// TwinCAT 3 PLC project IO_Main_Task
// ProgramVersion: 3.1.4026.19
// libraries:
//   Tc2_Standard, * (Beckhoff Automation GmbH)
//   Tc2_System, * (Beckhoff Automation GmbH)
//   Tc3_Module, * (Beckhoff Automation GmbH)
// project tree:
//   DUTs/EtherCAT模組/ EL1409.TcDUT, Murr_IMPACT67.TcDUT, EL2409.TcDUT
//   DUTs/ In_16_To_PLC.TcDUT, Out_16_To_PLC.TcDUT
//   GVLs/ EtherCAT.TcGVL, MainIO.TcGVL
//   / IO_Task.TcTTO
//   POUs/IO轉換/ AI_force.TcPOU, IO_force.TcPOU
//   POUs/IO轉換/控制櫃/ Mod101.TcPOU, Mod401.TcPOU, Mod102.TcPOU, Mod103.TcPOU, Mod104.TcPOU, Mod105.TcPOU, Mod106.TcPOU, Mod107.TcPOU, Mod108.TcPOU, Mod109.TcPOU
//   POUs/ MAIN.TcPOU
// (motion and I/O tree: see PLC project main)
// real-time tasks:
//   TASK Main_IO_Task: cycle T#2ms, priority 6, ADS port 353
//   TASK PlcTask: cycle T#10ms, priority 14, ADS port 350
//   TASK Conveyor: cycle T#10ms, priority 22, ADS port 355
// variable links:

CONFIGURATION IO_Main_Task
    RESOURCE PLC ON TwinCAT3
        TASK IO_Task(INTERVAL := T#2ms, PRIORITY := 6);
        PROGRAM MAIN WITH IO_Task : MAIN;
    END_RESOURCE
END_CONFIGURATION

// ---- DUTs/EtherCAT模組/EL1409.TcDUT
TYPE EL1409 :
STRUCT
	ModType : STRING := 'EL1409';
	Input AT %I*:ARRAY [1..16] OF BOOL;
	WcState AT %I*:BOOL;
	InputToggle AT %I*:BOOL;
	State AT %I*:UINT;
END_STRUCT
END_TYPE

// ---- DUTs/EtherCAT模組/Murr_IMPACT67.TcDUT
TYPE Murr_IMPACT67 :
STRUCT
	ModType : STRING := 'Murr IMPACT67';
	
	Input AT %I*:UINT;
	
	Output AT %Q*:UINT;
	
	Io_State AT %I*:ARRAY[0..7] OF USINT;
	
	WcState AT %I*:BOOL;
	InputToggle AT %I*:BOOL;
	State AT %I*:UINT;
END_STRUCT
END_TYPE

// ---- DUTs/EtherCAT模組/EL2409.TcDUT
TYPE EL2409 :
STRUCT
	ModType : STRING := 'EL2409';
	WcState AT %I*:BOOL;
	State AT %I*:UINT;
	
	Output AT %Q*:ARRAY [1..16] OF BOOL;
END_STRUCT
END_TYPE

// ---- DUTs/In_16_To_PLC.TcDUT
TYPE In_16_To_PLC :
STRUCT
	In AT %Q*:ARRAY [1..16] OF BOOL;
END_STRUCT
END_TYPE

// ---- DUTs/Out_16_To_PLC.TcDUT
TYPE Out_16_To_PLC :
STRUCT
	Out AT %I*:ARRAY [1..16] OF BOOL;
END_STRUCT
END_TYPE

// ---- GVLs/EtherCAT.TcGVL
{attribute 'qualified_only'}
VAR_GLOBAL
	// 主控制櫃 控制器
	MainMod_1 :EL1409;
	MainMod_2 :EL1409;
	MainMod_3 :EL1409;
	MainMod_4 :EL1409;
	MainMod_5 :EL1409;
	MainMod_6 :EL1409;
	MainMod_7 :EL2409;
	MainMod_8 :EL2409;
	MainMod_9 :EL2409;
	
	Murr_Mod : Murr_IMPACT67;
END_VAR

// ---- GVLs/MainIO.TcGVL
{attribute 'qualified_onlY0'}
VAR_GLOBAL
	//
	IO101: In_16_To_PLC;
	//
	IO102: In_16_To_PLC;
	//
	IO103: In_16_To_PLC;
	//
	IO104: In_16_To_PLC;
	//
	IO105: In_16_To_PLC;
	//
	IO106: In_16_To_PLC;
	//
	IO107: Out_16_To_PLC;
	//
	IO108: Out_16_To_PLC;
	//
	IO109: Out_16_To_PLC;
	
	//
	IO401: In_16_To_PLC;
	

	IO101_s : WORD;
	IO102_s : WORD;
	IO103_s : WORD;
	IO104_s : WORD;
	IO105_s : WORD;
	IO106_s : WORD;
	IO107_s : WORD;
	IO108_s : WORD;
	IO109_s : WORD;
	
	IO401_s : WORD;
	
	IO101_f : WORD;
	IO102_f : WORD;
	IO103_f : WORD;
	IO104_f : WORD;
	IO105_f : WORD;
	IO106_f : WORD;
	IO107_f : WORD;
	IO108_f : WORD;
	IO109_f : WORD;
	
	IO401_f : WORD;
END_VAR

// ---- POUs/MAIN.TcPOU
PROGRAM MAIN
VAR

END_VAR

Mod101();
Mod102();
Mod103();
Mod104();
Mod105();
Mod106();
Mod107();
Mod108();
Mod109();

Mod401();

END_PROGRAM

// ---- POUs/IO轉換/控制櫃/Mod101.TcPOU
PROGRAM Mod101
VAR
	IO_f : ARRAY [1..16] OF IO_force;
	
	i: SINT;
END_VAR

	// 輸入模組1
	FOR i := 1 TO 16 DO
		IO_f[i](Raw_IO := EtherCAT.MainMod_1.Input[i], Out =>MainIO.IO101.In[i]);
	END_FOR
	
	
	MainIO.IO101_s.0 := IO_f[1].Out;
	MainIO.IO101_s.1 := IO_f[2].Out;
	MainIO.IO101_s.2 := IO_f[3].Out;
	MainIO.IO101_s.3 := IO_f[4].Out;
	MainIO.IO101_s.4 := IO_f[5].Out;
	MainIO.IO101_s.5 := IO_f[6].Out;
	MainIO.IO101_s.6 := IO_f[7].Out;
	MainIO.IO101_s.7 := IO_f[8].Out;
	MainIO.IO101_s.8 := IO_f[9].Out;
	MainIO.IO101_s.9 := IO_f[10].Out;
	MainIO.IO101_s.10 := IO_f[11].Out;
	MainIO.IO101_s.11 := IO_f[12].Out;
	MainIO.IO101_s.12 := IO_f[13].Out;
	MainIO.IO101_s.13 := IO_f[14].Out;
	MainIO.IO101_s.14 := IO_f[15].Out;
	MainIO.IO101_s.15 := IO_f[16].Out;
	
	MainIO.io101_f.0 := IO_f[1].ForceEnable;
	MainIO.io101_f.1 := IO_f[2].ForceEnable;
	MainIO.io101_f.2 := IO_f[3].ForceEnable;
	MainIO.io101_f.3 := IO_f[4].ForceEnable;
	MainIO.io101_f.4 := IO_f[5].ForceEnable;
	MainIO.io101_f.5 := IO_f[6].ForceEnable;
	MainIO.io101_f.6 := IO_f[7].ForceEnable;
	MainIO.io101_f.7 := IO_f[8].ForceEnable;
	MainIO.io101_f.8 := IO_f[9].ForceEnable;
	MainIO.io101_f.9 := IO_f[10].ForceEnable;
	MainIO.io101_f.10 := IO_f[11].ForceEnable;
	MainIO.io101_f.11 := IO_f[12].ForceEnable;
	MainIO.io101_f.12 := IO_f[13].ForceEnable;
	MainIO.io101_f.13 := IO_f[14].ForceEnable;
	MainIO.io101_f.14 := IO_f[15].ForceEnable;
	MainIO.io101_f.15 := IO_f[16].ForceEnable;

END_PROGRAM

// ---- POUs/IO轉換/IO_force.TcPOU
FUNCTION_BLOCK IO_force
VAR_INPUT
	Raw_IO : BOOL;
END_VAR

VAR_OUTPUT
	Out : BOOL;
END_VAR

VAR
	ForceEnable : BOOL;
	ForceStatus : BOOL;
END_VAR

IF NOT ForceEnable THEN
	OUT := Raw_IO;
ELSE
	OUT := ForceStatus;
END_IF

END_FUNCTION_BLOCK

// ---- POUs/IO轉換/控制櫃/Mod102.TcPOU
PROGRAM Mod102
VAR
	IO_f : ARRAY [1..16] OF IO_force;
	i: SINT;
END_VAR

	// 輸入模組1
	FOR i := 1 TO 16 DO
		IO_f[i](Raw_IO := EtherCAT.MainMod_2.Input[i], Out =>MainIO.io102.In[i]);
	END_FOR
	
	
	MainIO.io102_s.0 := IO_f[1].Out;
	MainIO.io102_s.1 := IO_f[2].Out;
	MainIO.io102_s.2 := IO_f[3].Out;
	MainIO.io102_s.3 := IO_f[4].Out;
	MainIO.io102_s.4 := IO_f[5].Out;
	MainIO.io102_s.5 := IO_f[6].Out;
	MainIO.io102_s.6 := IO_f[7].Out;
	MainIO.io102_s.7 := IO_f[8].Out;
	MainIO.io102_s.8 := IO_f[9].Out;
	MainIO.io102_s.9 := IO_f[10].Out;
	MainIO.io102_s.10 := IO_f[11].Out;
	MainIO.io102_s.11 := IO_f[12].Out;
	MainIO.io102_s.12 := IO_f[13].Out;
	MainIO.io102_s.13 := IO_f[14].Out;
	MainIO.io102_s.14 := IO_f[15].Out;
	MainIO.io102_s.15 := IO_f[16].Out;
	
	MainIO.io102_f.0 := IO_f[1].ForceEnable;
	MainIO.io102_f.1 := IO_f[2].ForceEnable;
	MainIO.io102_f.2 := IO_f[3].ForceEnable;
	MainIO.io102_f.3 := IO_f[4].ForceEnable;
	MainIO.io102_f.4 := IO_f[5].ForceEnable;
	MainIO.io102_f.5 := IO_f[6].ForceEnable;
	MainIO.io102_f.6 := IO_f[7].ForceEnable;
	MainIO.io102_f.7 := IO_f[8].ForceEnable;
	MainIO.io102_f.8 := IO_f[9].ForceEnable;
	MainIO.io102_f.9 := IO_f[10].ForceEnable;
	MainIO.io102_f.10 := IO_f[11].ForceEnable;
	MainIO.io102_f.11 := IO_f[12].ForceEnable;
	MainIO.io102_f.12 := IO_f[13].ForceEnable;
	MainIO.io102_f.13 := IO_f[14].ForceEnable;
	MainIO.io102_f.14 := IO_f[15].ForceEnable;
	MainIO.io102_f.15 := IO_f[16].ForceEnable;

END_PROGRAM

// ---- POUs/IO轉換/控制櫃/Mod103.TcPOU
PROGRAM Mod103
VAR
	IO_f : ARRAY [1..16] OF IO_force;
	i: SINT;
END_VAR

	// 輸入模組1
	FOR i := 1 TO 16 DO
		IO_f[i](Raw_IO := EtherCAT.MainMod_3.Input[i], Out =>MainIO.io103.In[i]);
	END_FOR
	
	
	MainIO.io103_s.0 := IO_f[1].Out;
	MainIO.io103_s.1 := IO_f[2].Out;
	MainIO.io103_s.2 := IO_f[3].Out;
	MainIO.io103_s.3 := IO_f[4].Out;
	MainIO.io103_s.4 := IO_f[5].Out;
	MainIO.io103_s.5 := IO_f[6].Out;
	MainIO.io103_s.6 := IO_f[7].Out;
	MainIO.io103_s.7 := IO_f[8].Out;
	MainIO.io103_s.8 := IO_f[9].Out;
	MainIO.io103_s.9 := IO_f[10].Out;
	MainIO.io103_s.10 := IO_f[11].Out;
	MainIO.io103_s.11 := IO_f[12].Out;
	MainIO.io103_s.12 := IO_f[13].Out;
	MainIO.io103_s.13 := IO_f[14].Out;
	MainIO.io103_s.14 := IO_f[15].Out;
	MainIO.io103_s.15 := IO_f[16].Out;
	
	MainIO.io103_f.0 := IO_f[1].ForceEnable;
	MainIO.io103_f.1 := IO_f[2].ForceEnable;
	MainIO.io103_f.2 := IO_f[3].ForceEnable;
	MainIO.io103_f.3 := IO_f[4].ForceEnable;
	MainIO.io103_f.4 := IO_f[5].ForceEnable;
	MainIO.io103_f.5 := IO_f[6].ForceEnable;
	MainIO.io103_f.6 := IO_f[7].ForceEnable;
	MainIO.io103_f.7 := IO_f[8].ForceEnable;
	MainIO.io103_f.8 := IO_f[9].ForceEnable;
	MainIO.io103_f.9 := IO_f[10].ForceEnable;
	MainIO.io103_f.10 := IO_f[11].ForceEnable;
	MainIO.io103_f.11 := IO_f[12].ForceEnable;
	MainIO.io103_f.12 := IO_f[13].ForceEnable;
	MainIO.io103_f.13 := IO_f[14].ForceEnable;
	MainIO.io103_f.14 := IO_f[15].ForceEnable;
	MainIO.io103_f.15 := IO_f[16].ForceEnable;

END_PROGRAM

// ---- POUs/IO轉換/控制櫃/Mod104.TcPOU
PROGRAM Mod104
VAR
	IO_f : ARRAY [1..16] OF IO_force;
	i: SINT;
END_VAR

	// 輸入模組1
	FOR i := 1 TO 16 DO
		IO_f[i](Raw_IO := EtherCAT.MainMod_4.Input[i], Out =>MainIO.io104.In[i]);
	END_FOR
	
	
	MainIO.io104_s.0 := IO_f[1].Out;
	MainIO.io104_s.1 := IO_f[2].Out;
	MainIO.io104_s.2 := IO_f[3].Out;
	MainIO.io104_s.3 := IO_f[4].Out;
	MainIO.io104_s.4 := IO_f[5].Out;
	MainIO.io104_s.5 := IO_f[6].Out;
	MainIO.io104_s.6 := IO_f[7].Out;
	MainIO.io104_s.7 := IO_f[8].Out;
	MainIO.io104_s.8 := IO_f[9].Out;
	MainIO.io104_s.9 := IO_f[10].Out;
	MainIO.io104_s.10 := IO_f[11].Out;
	MainIO.io104_s.11 := IO_f[12].Out;
	MainIO.io104_s.12 := IO_f[13].Out;
	MainIO.io104_s.13 := IO_f[14].Out;
	MainIO.io104_s.14 := IO_f[15].Out;
	MainIO.io104_s.15 := IO_f[16].Out;
	
	MainIO.io104_f.0 := IO_f[1].ForceEnable;
	MainIO.io104_f.1 := IO_f[2].ForceEnable;
	MainIO.io104_f.2 := IO_f[3].ForceEnable;
	MainIO.io104_f.3 := IO_f[4].ForceEnable;
	MainIO.io104_f.4 := IO_f[5].ForceEnable;
	MainIO.io104_f.5 := IO_f[6].ForceEnable;
	MainIO.io104_f.6 := IO_f[7].ForceEnable;
	MainIO.io104_f.7 := IO_f[8].ForceEnable;
	MainIO.io104_f.8 := IO_f[9].ForceEnable;
	MainIO.io104_f.9 := IO_f[10].ForceEnable;
	MainIO.io104_f.10 := IO_f[11].ForceEnable;
	MainIO.io104_f.11 := IO_f[12].ForceEnable;
	MainIO.io104_f.12 := IO_f[13].ForceEnable;
	MainIO.io104_f.13 := IO_f[14].ForceEnable;
	MainIO.io104_f.14 := IO_f[15].ForceEnable;
	MainIO.io104_f.15 := IO_f[16].ForceEnable;

END_PROGRAM

// ---- POUs/IO轉換/控制櫃/Mod105.TcPOU
PROGRAM Mod105
VAR
	IO_f : ARRAY [1..16] OF IO_force;
	i: SINT;
END_VAR

	// 輸入模組1
	FOR i := 1 TO 16 DO
		IO_f[i](Raw_IO := EtherCAT.MainMod_5.Input[i], Out =>MainIO.io105.In[i]);
	END_FOR
	
	
	MainIO.io105_s.0 := IO_f[1].Out;
	MainIO.io105_s.1 := IO_f[2].Out;
	MainIO.io105_s.2 := IO_f[3].Out;
	MainIO.io105_s.3 := IO_f[4].Out;
	MainIO.io105_s.4 := IO_f[5].Out;
	MainIO.io105_s.5 := IO_f[6].Out;
	MainIO.io105_s.6 := IO_f[7].Out;
	MainIO.io105_s.7 := IO_f[8].Out;
	MainIO.io105_s.8 := IO_f[9].Out;
	MainIO.io105_s.9 := IO_f[10].Out;
	MainIO.io105_s.10 := IO_f[11].Out;
	MainIO.io105_s.11 := IO_f[12].Out;
	MainIO.io105_s.12 := IO_f[13].Out;
	MainIO.io105_s.13 := IO_f[14].Out;
	MainIO.io105_s.14 := IO_f[15].Out;
	MainIO.io105_s.15 := IO_f[16].Out;
	
	MainIO.io105_f.0 := IO_f[1].ForceEnable;
	MainIO.io105_f.1 := IO_f[2].ForceEnable;
	MainIO.io105_f.2 := IO_f[3].ForceEnable;
	MainIO.io105_f.3 := IO_f[4].ForceEnable;
	MainIO.io105_f.4 := IO_f[5].ForceEnable;
	MainIO.io105_f.5 := IO_f[6].ForceEnable;
	MainIO.io105_f.6 := IO_f[7].ForceEnable;
	MainIO.io105_f.7 := IO_f[8].ForceEnable;
	MainIO.io105_f.8 := IO_f[9].ForceEnable;
	MainIO.io105_f.9 := IO_f[10].ForceEnable;
	MainIO.io105_f.10 := IO_f[11].ForceEnable;
	MainIO.io105_f.11 := IO_f[12].ForceEnable;
	MainIO.io105_f.12 := IO_f[13].ForceEnable;
	MainIO.io105_f.13 := IO_f[14].ForceEnable;
	MainIO.io105_f.14 := IO_f[15].ForceEnable;
	MainIO.io105_f.15 := IO_f[16].ForceEnable;

END_PROGRAM

// ---- POUs/IO轉換/控制櫃/Mod106.TcPOU
PROGRAM Mod106
VAR
	IO_f : ARRAY [1..16] OF IO_force;
	i: SINT;
END_VAR

	// 輸入模組1
	FOR i := 1 TO 16 DO
		IO_f[i](Raw_IO := EtherCAT.MainMod_6.Input[i], Out =>MainIO.io106.In[i]);
	END_FOR
	
	
	MainIO.io106_s.0 := IO_f[1].Out;
	MainIO.io106_s.1 := IO_f[2].Out;
	MainIO.io106_s.2 := IO_f[3].Out;
	MainIO.io106_s.3 := IO_f[4].Out;
	MainIO.io106_s.4 := IO_f[5].Out;
	MainIO.io106_s.5 := IO_f[6].Out;
	MainIO.io106_s.6 := IO_f[7].Out;
	MainIO.io106_s.7 := IO_f[8].Out;
	MainIO.io106_s.8 := IO_f[9].Out;
	MainIO.io106_s.9 := IO_f[10].Out;
	MainIO.io106_s.10 := IO_f[11].Out;
	MainIO.io106_s.11 := IO_f[12].Out;
	MainIO.io106_s.12 := IO_f[13].Out;
	MainIO.io106_s.13 := IO_f[14].Out;
	MainIO.io106_s.14 := IO_f[15].Out;
	MainIO.io106_s.15 := IO_f[16].Out;
	
	MainIO.io106_f.0 := IO_f[1].ForceEnable;
	MainIO.io106_f.1 := IO_f[2].ForceEnable;
	MainIO.io106_f.2 := IO_f[3].ForceEnable;
	MainIO.io106_f.3 := IO_f[4].ForceEnable;
	MainIO.io106_f.4 := IO_f[5].ForceEnable;
	MainIO.io106_f.5 := IO_f[6].ForceEnable;
	MainIO.io106_f.6 := IO_f[7].ForceEnable;
	MainIO.io106_f.7 := IO_f[8].ForceEnable;
	MainIO.io106_f.8 := IO_f[9].ForceEnable;
	MainIO.io106_f.9 := IO_f[10].ForceEnable;
	MainIO.io106_f.10 := IO_f[11].ForceEnable;
	MainIO.io106_f.11 := IO_f[12].ForceEnable;
	MainIO.io106_f.12 := IO_f[13].ForceEnable;
	MainIO.io106_f.13 := IO_f[14].ForceEnable;
	MainIO.io106_f.14 := IO_f[15].ForceEnable;
	MainIO.io106_f.15 := IO_f[16].ForceEnable;

END_PROGRAM

// ---- POUs/IO轉換/控制櫃/Mod107.TcPOU
PROGRAM Mod107
VAR
	IO_f : ARRAY [1..16] OF IO_force;
	
	i: SINT;
END_VAR

	// 輸入模組1
	FOR i := 1 TO 16 DO
		IO_f[i](Raw_IO := MainIO.IO107.Out[i], Out => EtherCAT.MainMod_7.Output[i]);
	END_FOR
	
	
	MainIO.IO107_s.0 := IO_f[1].Out;
	MainIO.IO107_s.1 := IO_f[2].Out;
	MainIO.IO107_s.2 := IO_f[3].Out;
	MainIO.IO107_s.3 := IO_f[4].Out;
	MainIO.IO107_s.4 := IO_f[5].Out;
	MainIO.IO107_s.5 := IO_f[6].Out;
	MainIO.IO107_s.6 := IO_f[7].Out;
	MainIO.IO107_s.7 := IO_f[8].Out;
	MainIO.IO107_s.8 := IO_f[9].Out;
	MainIO.IO107_s.9 := IO_f[10].Out;
	MainIO.IO107_s.10 := IO_f[11].Out;
	MainIO.IO107_s.11 := IO_f[12].Out;
	MainIO.IO107_s.12 := IO_f[13].Out;
	MainIO.IO107_s.13 := IO_f[14].Out;
	MainIO.IO107_s.14 := IO_f[15].Out;
	MainIO.IO107_s.15 := IO_f[16].Out;
	
	MainIO.IO107_f.0 := IO_f[1].ForceEnable;
	MainIO.IO107_f.1 := IO_f[2].ForceEnable;
	MainIO.IO107_f.2 := IO_f[3].ForceEnable;
	MainIO.IO107_f.3 := IO_f[4].ForceEnable;
	MainIO.IO107_f.4 := IO_f[5].ForceEnable;
	MainIO.IO107_f.5 := IO_f[6].ForceEnable;
	MainIO.IO107_f.6 := IO_f[7].ForceEnable;
	MainIO.IO107_f.7 := IO_f[8].ForceEnable;
	MainIO.IO107_f.8 := IO_f[9].ForceEnable;
	MainIO.IO107_f.9 := IO_f[10].ForceEnable;
	MainIO.IO107_f.10 := IO_f[11].ForceEnable;
	MainIO.IO107_f.11 := IO_f[12].ForceEnable;
	MainIO.IO107_f.12 := IO_f[13].ForceEnable;
	MainIO.IO107_f.13 := IO_f[14].ForceEnable;
	MainIO.IO107_f.14 := IO_f[15].ForceEnable;
	MainIO.IO107_f.15 := IO_f[16].ForceEnable;

END_PROGRAM

// ---- POUs/IO轉換/控制櫃/Mod108.TcPOU
PROGRAM Mod108
VAR
	IO_f : ARRAY [1..16] OF IO_force;
	
	i: SINT;
END_VAR

	// 輸入模組1
	FOR i := 1 TO 16 DO
		IO_f[i](Raw_IO := MainIO.IO108.Out[i], Out => EtherCAT.MainMod_8.Output[i]);
	END_FOR
	
	
	MainIO.IO108_s.0 := IO_f[1].Out;
	MainIO.IO108_s.1 := IO_f[2].Out;
	MainIO.IO108_s.2 := IO_f[3].Out;
	MainIO.IO108_s.3 := IO_f[4].Out;
	MainIO.IO108_s.4 := IO_f[5].Out;
	MainIO.IO108_s.5 := IO_f[6].Out;
	MainIO.IO108_s.6 := IO_f[7].Out;
	MainIO.IO108_s.7 := IO_f[8].Out;
	MainIO.IO108_s.8 := IO_f[9].Out;
	MainIO.IO108_s.9 := IO_f[10].Out;
	MainIO.IO108_s.10 := IO_f[11].Out;
	MainIO.IO108_s.11 := IO_f[12].Out;
	MainIO.IO108_s.12 := IO_f[13].Out;
	MainIO.IO108_s.13 := IO_f[14].Out;
	MainIO.IO108_s.14 := IO_f[15].Out;
	MainIO.IO108_s.15 := IO_f[16].Out;
	
	MainIO.IO108_f.0 := IO_f[1].ForceEnable;
	MainIO.IO108_f.1 := IO_f[2].ForceEnable;
	MainIO.IO108_f.2 := IO_f[3].ForceEnable;
	MainIO.IO108_f.3 := IO_f[4].ForceEnable;
	MainIO.IO108_f.4 := IO_f[5].ForceEnable;
	MainIO.IO108_f.5 := IO_f[6].ForceEnable;
	MainIO.IO108_f.6 := IO_f[7].ForceEnable;
	MainIO.IO108_f.7 := IO_f[8].ForceEnable;
	MainIO.IO108_f.8 := IO_f[9].ForceEnable;
	MainIO.IO108_f.9 := IO_f[10].ForceEnable;
	MainIO.IO108_f.10 := IO_f[11].ForceEnable;
	MainIO.IO108_f.11 := IO_f[12].ForceEnable;
	MainIO.IO108_f.12 := IO_f[13].ForceEnable;
	MainIO.IO108_f.13 := IO_f[14].ForceEnable;
	MainIO.IO108_f.14 := IO_f[15].ForceEnable;
	MainIO.IO108_f.15 := IO_f[16].ForceEnable;

END_PROGRAM

// ---- POUs/IO轉換/控制櫃/Mod109.TcPOU
PROGRAM Mod109
VAR
	IO_f : ARRAY [1..16] OF IO_force;
	
	i: SINT;
END_VAR

	// 輸入模組1
	FOR i := 1 TO 16 DO
		IO_f[i](Raw_IO := MainIO.IO109.Out[i], Out => EtherCAT.MainMod_9.Output[i]);
	END_FOR
	
	
	MainIO.IO109_s.0 := IO_f[1].Out;
	MainIO.IO109_s.1 := IO_f[2].Out;
	MainIO.IO109_s.2 := IO_f[3].Out;
	MainIO.IO109_s.3 := IO_f[4].Out;
	MainIO.IO109_s.4 := IO_f[5].Out;
	MainIO.IO109_s.5 := IO_f[6].Out;
	MainIO.IO109_s.6 := IO_f[7].Out;
	MainIO.IO109_s.7 := IO_f[8].Out;
	MainIO.IO109_s.8 := IO_f[9].Out;
	MainIO.IO109_s.9 := IO_f[10].Out;
	MainIO.IO109_s.10 := IO_f[11].Out;
	MainIO.IO109_s.11 := IO_f[12].Out;
	MainIO.IO109_s.12 := IO_f[13].Out;
	MainIO.IO109_s.13 := IO_f[14].Out;
	MainIO.IO109_s.14 := IO_f[15].Out;
	MainIO.IO109_s.15 := IO_f[16].Out;
	
	MainIO.IO109_f.0 := IO_f[1].ForceEnable;
	MainIO.IO109_f.1 := IO_f[2].ForceEnable;
	MainIO.IO109_f.2 := IO_f[3].ForceEnable;
	MainIO.IO109_f.3 := IO_f[4].ForceEnable;
	MainIO.IO109_f.4 := IO_f[5].ForceEnable;
	MainIO.IO109_f.5 := IO_f[6].ForceEnable;
	MainIO.IO109_f.6 := IO_f[7].ForceEnable;
	MainIO.IO109_f.7 := IO_f[8].ForceEnable;
	MainIO.IO109_f.8 := IO_f[9].ForceEnable;
	MainIO.IO109_f.9 := IO_f[10].ForceEnable;
	MainIO.IO109_f.10 := IO_f[11].ForceEnable;
	MainIO.IO109_f.11 := IO_f[12].ForceEnable;
	MainIO.IO109_f.12 := IO_f[13].ForceEnable;
	MainIO.IO109_f.13 := IO_f[14].ForceEnable;
	MainIO.IO109_f.14 := IO_f[15].ForceEnable;
	MainIO.IO109_f.15 := IO_f[16].ForceEnable;

END_PROGRAM

// ---- POUs/IO轉換/控制櫃/Mod401.TcPOU
PROGRAM Mod401
VAR
	ioRawWord :WORD;

	ioRaw : ARRAY [1..16] OF BOOL;

	IO_f : ARRAY [1..16] OF IO_force;
	
	i: SINT;
END_VAR

conver();
	// 輸入模組1
	FOR i := 1 TO 16 DO
		IO_f[i](Raw_IO := ioRaw[i], Out =>MainIO.IO401.In[i]);
	END_FOR
	
	
	MainIO.IO401_s.0 := IO_f[1].Out;
	MainIO.IO401_s.1 := IO_f[2].Out;
	MainIO.IO401_s.2 := IO_f[3].Out;
	MainIO.IO401_s.3 := IO_f[4].Out;
	MainIO.IO401_s.4 := IO_f[5].Out;
	MainIO.IO401_s.5 := IO_f[6].Out;
	MainIO.IO401_s.6 := IO_f[7].Out;
	MainIO.IO401_s.7 := IO_f[8].Out;
	MainIO.IO401_s.8 := IO_f[9].Out;
	MainIO.IO401_s.9 := IO_f[10].Out;
	MainIO.IO401_s.10 := IO_f[11].Out;
	MainIO.IO401_s.11 := IO_f[12].Out;
	MainIO.IO401_s.12 := IO_f[13].Out;
	MainIO.IO401_s.13 := IO_f[14].Out;
	MainIO.IO401_s.14 := IO_f[15].Out;
	MainIO.IO401_s.15 := IO_f[16].Out;
	
	MainIO.IO401_f.0 := IO_f[1].ForceEnable;
	MainIO.IO401_f.1 := IO_f[2].ForceEnable;
	MainIO.IO401_f.2 := IO_f[3].ForceEnable;
	MainIO.IO401_f.3 := IO_f[4].ForceEnable;
	MainIO.IO401_f.4 := IO_f[5].ForceEnable;
	MainIO.IO401_f.5 := IO_f[6].ForceEnable;
	MainIO.IO401_f.6 := IO_f[7].ForceEnable;
	MainIO.IO401_f.7 := IO_f[8].ForceEnable;
	MainIO.IO401_f.8 := IO_f[9].ForceEnable;
	MainIO.IO401_f.9 := IO_f[10].ForceEnable;
	MainIO.IO401_f.10 := IO_f[11].ForceEnable;
	MainIO.IO401_f.11 := IO_f[12].ForceEnable;
	MainIO.IO401_f.12 := IO_f[13].ForceEnable;
	MainIO.IO401_f.13 := IO_f[14].ForceEnable;
	MainIO.IO401_f.14 := IO_f[15].ForceEnable;
	MainIO.IO401_f.15 := IO_f[16].ForceEnable;

ACTION conver:
ioRawWord := TO_WORD(EtherCAT.Murr_Mod.Input);
	
ioRaw[1] := ioRawWord.0;
ioRaw[2] := ioRawWord.1;
ioRaw[3] := ioRawWord.2;
ioRaw[4] := ioRawWord.3;
ioRaw[5] := ioRawWord.4;
ioRaw[6] := ioRawWord.5;
ioRaw[7] := ioRawWord.6;
ioRaw[8] := ioRawWord.7;
ioRaw[9] := ioRawWord.8;
ioRaw[10] := ioRawWord.9;
ioRaw[11] := ioRawWord.10;
ioRaw[12] := ioRawWord.11;
ioRaw[13] := ioRawWord.12;
ioRaw[14] := ioRawWord.13;
ioRaw[15] := ioRawWord.14;
ioRaw[16] := ioRawWord.15;
END_ACTION

END_PROGRAM

// ---- POUs/IO轉換/AI_force.TcPOU
FUNCTION_BLOCK AI_force
VAR_INPUT
	Raw_IO : INT;
END_VAR

VAR_OUTPUT
	Out : INT;
END_VAR

VAR
	ForceEnable : BOOL;
	ForceValue : INT;
END_VAR

IF NOT ForceEnable THEN
	OUT := Raw_IO;
ELSE
	OUT := ForceValue;
END_IF

END_FUNCTION_BLOCK
